// TwinCAT 3 PLC project Tc3_CRC
// Title: Tc3_CRC
// Company: RKe
// Author: Kim Robbens
// ProjectVersion: 0.0.0.2
// Description: CRC (Cyclic Redundancy Check) calculation with support for numerous standard CRC algorithms
// ProgramVersion: 3.1.4026.17
// libraries:
//   Tc2_Utilities, * (Beckhoff Automation GmbH)
//   Tc3_AlgoInterfaces, * (RKe)
// project tree:
//   DUTs/ E_CRC_Mode.TcDUT, E_CRC_Type.TcDUT, ST_CRC_Params.TcDUT, U_8BYTEARRAY.TcDUT
//   GVCs/ GVC_CRC.TcGVL
//   POUs/ CRC.TcPOU
//   Project Information/ F_GetCompany.TcPOU, F_GetTitle.TcPOU, F_GetVersion.TcPOU
//   Version/ Global_Version.TcGVL

// ---- DUTs/E_CRC_Mode.TcDUT
{attribute 'qualified_only'}
{attribute 'strict'}
{attribute 'to_string'}
TYPE E_CRC_Mode :
(
	CRC8	:= 0,
	CRC16 	:= 1,
	CRC24 	:= 2,
	CRC32 	:= 3,
	CRC40 	:= 4,
	CRC64 	:= 7
) BYTE;
END_TYPE

// ---- DUTs/E_CRC_Type.TcDUT
{attribute 'qualified_only'}
{attribute 'to_string'}
TYPE E_CRC_Type : (
    CRC_8_AUTOSAR,
    CRC_8_BLUETOOTH,
    CRC_8_CDMA2000,
    CRC_8_DARC,
    CRC_8_DVB_S2,
    CRC_8_GSM_A,
    CRC_8_GSM_B,
    CRC_8_HITAG,
    CRC_8_I_432_1,
    CRC_8_I_CODE,
    CRC_8_LTE,
    CRC_8_MAXIM_DOW,
    CRC_8_MIFARE_MAD,
    CRC_8_NRSC_5,
    CRC_8_OPENSAFETY,
    CRC_8_ROHC,
    CRC_8_SAE_J1850,
    CRC_8_SMBUS,
    CRC_8_TECH_3250,
    CRC_8_WCDMA,
    CRC_16_ARC,
    CRC_16_CDMA2000,
    CRC_16_CMS,
    CRC_16_DDS_110,
    CRC_16_DECT_R,
    CRC_16_DECT_X,
    CRC_16_DNP,
    CRC_16_EN_13757,
    CRC_16_GENIBUS,
    CRC_16_GSM,
    CRC_16_IBM_3740,
    CRC_16_IBM_SDLC,
    CRC_16_ISO_IEC_14443_3_A,
    CRC_16_KERMIT,
    CRC_16_LJ1200,
    CRC_16_MAXIM_DOW,
    CRC_16_MCRF4XX,
    CRC_16_MODBUS,
    CRC_16_NRSC_5,
    CRC_16_OPENSAFETY_A,
    CRC_16_OPENSAFETY_B,
    CRC_16_PROFIBUS,
    CRC_16_RIELLO,
    CRC_16_SPI_FUJITSU,
    CRC_16_T10_DIF,
    CRC_16_TELEDISK,
    CRC_16_TMS37157,
    CRC_16_UMTS,
    CRC_16_USB,
    CRC_16_XMODEM,
    CRC_24_BLE,
    CRC_24_FLEXRAY_A,
    CRC_24_FLEXRAY_B,
    CRC_24_INTERLAKEN,
    CRC_24_LTE_A,
    CRC_24_LTE_B,
    CRC_24_OPENPGP,
    CRC_24_OS_9,
    CRC_32_AIXM,
    CRC_32_AUTOSAR,
    CRC_32_BASE91_D,
    CRC_32_BZIP2,
    CRC_32_CD_ROM_EDC,
    CRC_32_CKSUM,
    CRC_32_ISCSI,
    CRC_32_ISO_HDLC,
    CRC_32_JAMCRC,
    CRC_32_MEF,
    CRC_32_MPEG_2,
    CRC_32_XFER,
    CRC_40_GSM,
    CRC_64_ECMA_182,
    CRC_64_GO_ISO,
    CRC_64_MS,
    CRC_64_WE,
    CRC_64_XZ,
	CRC_NO_OF_TYPES  		// end of enum list placeholder
)BYTE;
END_TYPE

// ---- DUTs/ST_CRC_Params.TcDUT
TYPE ST_CRC_Params :
STRUCT
    bitWidth      		: BYTE;
    polynomial       	: XWORD;
    initCRC       		: XWORD;
    reflectInitial      : BOOL;
    reflected     		: BOOL;
    xorOut     			: XWORD;
    check      			: XWORD;
    residue    			: XWORD;
END_STRUCT
END_TYPE

// ---- DUTs/U_8BYTEARRAY.TcDUT
TYPE U_8BYTEARRAY :
UNION
	byteArray					: ARRAY[0..7] OF BYTE;
	xword_						: XWORD;
	dword_						: ARRAY[0..1] OF DWORD;					
	word_						: ARRAY[0..3] OF WORD;					
END_UNION
END_TYPE

// ---- GVCs/GVC_CRC.TcGVL
{attribute 'qualified_only'}
VAR_GLOBAL CONSTANT
	CRCMasks 		: ARRAY[0..E_CRC_Mode.CRC64] OF XWORD 	:= [16#FF, 16#FFFF, 16#FFFFFF, 16#FFFFFFFF, 16#FFFFFFFFFF, 16#0, 16#0, 16#FFFFFFFFFFFFFFFF];
	CRCMsb			: ARRAY[0..E_CRC_Mode.CRC64] OF XWORD 	:= [16#80, 16#8000, 16#800000, 16#80000000, 16#8000000000, 16#0, 16#0, 16#8000000000000000]; 
	CRCShift		: ARRAY[0..E_CRC_Mode.CRC64] OF BYTE 	:= [0, 8, 16, 24, 32, 0, 0, 56];	
	referenceCheck	: ARRAY[1..9] OF BYTE := [16#31, 16#32, 16#33, 16#34, 16#35, 16#36, 16#37, 16#38, 16#39]; // Number 123456789  

	// CRC Type definition
	// source: https://reveng.sourceforge.io/crc-catalogue/all.htm
	CRC_Parameters : ARRAY[0..E_CRC_Type.CRC_NO_OF_TYPES] OF ST_CRC_Params := [
(* CRC_8_AUTOSAR *)      		(bitWidth := 8, polynomial := 16#2F, initCRC := 16#FF, reflectInitial := FALSE, reflected := FALSE, XorOut := 16#FF, Check := 16#DF, Residue := 16#42),
(* CRC_8_BLUETOOTH *)    		(bitWidth := 8, polynomial := 16#A7, initCRC := 16#00, reflectInitial := FALSE, reflected := TRUE,  XorOut := 16#00, Check := 16#26, Residue := 16#00),
(* CRC_8_CDMA2000 *)     		(bitWidth := 8, polynomial := 16#9B, initCRC := 16#FF, reflectInitial := FALSE, reflected := FALSE, XorOut := 16#00, Check := 16#DA, Residue := 16#00),
(* CRC_8_DARC *)         		(bitWidth := 8, polynomial := 16#39, initCRC := 16#00, reflectInitial := FALSE, reflected := TRUE,  XorOut := 16#00, Check := 16#15, Residue := 16#00),
(* CRC_8_DVB_S2 *)       		(bitWidth := 8, polynomial := 16#D5, initCRC := 16#00, reflectInitial := FALSE, reflected := FALSE, XorOut := 16#00, Check := 16#BC, Residue := 16#00),
(* CRC_8_GSM_A *)        		(bitWidth := 8, polynomial := 16#1D, initCRC := 16#00, reflectInitial := FALSE, reflected := FALSE, XorOut := 16#00, Check := 16#37, Residue := 16#00),
(* CRC_8_GSM_B *)        		(bitWidth := 8, polynomial := 16#49, initCRC := 16#00, reflectInitial := FALSE, reflected := FALSE, XorOut := 16#FF, Check := 16#94, Residue := 16#53),
(* CRC_8_HITAG *)        		(bitWidth := 8, polynomial := 16#1D, initCRC := 16#FF, reflectInitial := FALSE, reflected := FALSE, XorOut := 16#00, Check := 16#B4, Residue := 16#00),
(* CRC_8_I_432_1 *)      		(bitWidth := 8, polynomial := 16#07, initCRC := 16#00, reflectInitial := FALSE, reflected := FALSE, XorOut := 16#55, Check := 16#A1, Residue := 16#AC),
(* CRC_8_I_CODE *)       		(bitWidth := 8, polynomial := 16#1D, initCRC := 16#FD, reflectInitial := FALSE, reflected := FALSE, XorOut := 16#00, Check := 16#7E, Residue := 16#00),
(* CRC_8_LTE *)          		(bitWidth := 8, polynomial := 16#9B, initCRC := 16#00, reflectInitial := FALSE, reflected := FALSE, XorOut := 16#00, Check := 16#EA, Residue := 16#00),
(* CRC_8_MAXIM_DOW *)    		(bitWidth := 8, polynomial := 16#31, initCRC := 16#00, reflectInitial := FALSE, reflected := TRUE,  XorOut := 16#00, Check := 16#A1, Residue := 16#00),
(* CRC_8_MIFARE_MAD *)   		(bitWidth := 8, polynomial := 16#1D, initCRC := 16#C7, reflectInitial := FALSE, reflected := FALSE, XorOut := 16#00, Check := 16#99, Residue := 16#00),
(* CRC_8_NRSC_5 *)       		(bitWidth := 8, polynomial := 16#31, initCRC := 16#FF, reflectInitial := FALSE, reflected := FALSE, XorOut := 16#00, Check := 16#F7, Residue := 16#00),
(* CRC_8_OPENSAFETY *)   		(bitWidth := 8, polynomial := 16#2F, initCRC := 16#00, reflectInitial := FALSE, reflected := FALSE, XorOut := 16#00, Check := 16#3E, Residue := 16#00),
(* CRC_8_ROHC *)         		(bitWidth := 8, polynomial := 16#07, initCRC := 16#FF, reflectInitial := FALSE, reflected := TRUE,  XorOut := 16#00, Check := 16#D0, Residue := 16#00),
(* CRC_8_SAE_J1850 *)    		(bitWidth := 8, polynomial := 16#1D, initCRC := 16#FF, reflectInitial := FALSE, reflected := FALSE, XorOut := 16#FF, Check := 16#4B, Residue := 16#C4),
(* CRC_8_SMBUS *)        		(bitWidth := 8, polynomial := 16#07, initCRC := 16#00, reflectInitial := FALSE, reflected := FALSE, XorOut := 16#00, Check := 16#F4, Residue := 16#00),
(* CRC_8_TECH_3250 *)    		(bitWidth := 8, polynomial := 16#1D, initCRC := 16#FF, reflectInitial := FALSE, reflected := TRUE,  XorOut := 16#00, Check := 16#97, Residue := 16#00),
(* CRC_8_WCDMA *)        		(bitWidth := 8, polynomial := 16#9B, initCRC := 16#00, reflectInitial := FALSE, reflected := TRUE,  XorOut := 16#00, Check := 16#25, Residue := 16#00),
(* CRC_16_ARC *)                (bitWidth := 16, polynomial := 16#8005, initCRC := 16#0000, reflectInitial := FALSE, reflected := TRUE,  XorOut := 16#0000, Check := 16#BB3D, Residue := 16#0000),
(* CRC_16_CDMA2000 *)           (bitWidth := 16, polynomial := 16#C867, initCRC := 16#FFFF, reflectInitial := FALSE, reflected := FALSE, XorOut := 16#0000, Check := 16#4C06, Residue := 16#0000),
(* CRC_16_CMS *)                (bitWidth := 16, polynomial := 16#8005, initCRC := 16#FFFF, reflectInitial := FALSE, reflected := FALSE, XorOut := 16#0000, Check := 16#AEE7, Residue := 16#0000),
(* CRC_16_DDS_110 *)            (bitWidth := 16, polynomial := 16#8005, initCRC := 16#800D, reflectInitial := FALSE, reflected := FALSE, XorOut := 16#0000, Check := 16#9ECF, Residue := 16#0000),
(* CRC_16_DECT_R *)             (bitWidth := 16, polynomial := 16#0589, initCRC := 16#0000, reflectInitial := FALSE, reflected := FALSE, XorOut := 16#0001, Check := 16#007E, Residue := 16#0589),
(* CRC_16_DECT_X *)             (bitWidth := 16, polynomial := 16#0589, initCRC := 16#0000, reflectInitial := FALSE, reflected := FALSE, XorOut := 16#0000, Check := 16#007F, Residue := 16#0000),
(* CRC_16_DNP *)                (bitWidth := 16, polynomial := 16#3D65, initCRC := 16#0000, reflectInitial := FALSE, reflected := TRUE,  XorOut := 16#FFFF, Check := 16#EA82, Residue := 16#66C5),
(* CRC_16_EN_13757 *)           (bitWidth := 16, polynomial := 16#3D65, initCRC := 16#0000, reflectInitial := FALSE, reflected := FALSE, XorOut := 16#FFFF, Check := 16#C2B7, Residue := 16#A366),
(* CRC_16_GENIBUS *)            (bitWidth := 16, polynomial := 16#1021, initCRC := 16#FFFF, reflectInitial := FALSE, reflected := FALSE, XorOut := 16#FFFF, Check := 16#D64E, Residue := 16#1D0F),
(* CRC_16_GSM *)                (bitWidth := 16, polynomial := 16#1021, initCRC := 16#0000, reflectInitial := FALSE, reflected := FALSE, XorOut := 16#FFFF, Check := 16#CE3C, Residue := 16#1D0F),
(* CRC_16_IBM_3740 *)           (bitWidth := 16, polynomial := 16#1021, initCRC := 16#FFFF, reflectInitial := FALSE, reflected := FALSE, XorOut := 16#0000, Check := 16#29B1, Residue := 16#0000),
(* CRC_16_IBM_SDLC *)           (bitWidth := 16, polynomial := 16#1021, initCRC := 16#FFFF, reflectInitial := FALSE, reflected := TRUE,  XorOut := 16#FFFF, Check := 16#906E, Residue := 16#F0B8),
(* CRC_16_ISO_IEC_14443_3_A *)  (bitWidth := 16, polynomial := 16#1021, initCRC := 16#C6C6, reflectInitial := TRUE,  reflected := TRUE,  XorOut := 16#0000, Check := 16#BF05, Residue := 16#0000),
(* CRC_16_KERMIT *)             (bitWidth := 16, polynomial := 16#1021, initCRC := 16#0000, reflectInitial := FALSE, reflected := TRUE,  XorOut := 16#0000, Check := 16#2189, Residue := 16#0000),
(* CRC_16_LJ1200 *)             (bitWidth := 16, polynomial := 16#6F63, initCRC := 16#0000, reflectInitial := FALSE, reflected := FALSE, XorOut := 16#0000, Check := 16#BDF4, Residue := 16#0000),
(* CRC_16_MAXIM_DOW *)          (bitWidth := 16, polynomial := 16#8005, initCRC := 16#0000, reflectInitial := FALSE, reflected := TRUE,  XorOut := 16#FFFF, Check := 16#44C2, Residue := 16#B001),
(* CRC_16_MCRF4XX *)            (bitWidth := 16, polynomial := 16#1021, initCRC := 16#FFFF, reflectInitial := FALSE, reflected := TRUE,  XorOut := 16#0000, Check := 16#6F91, Residue := 16#0000),
(* CRC_16_MODBUS *)             (bitWidth := 16, polynomial := 16#8005, initCRC := 16#FFFF, reflectInitial := FALSE, reflected := TRUE,  XorOut := 16#0000, Check := 16#4B37, Residue := 16#0000),
(* CRC_16_NRSC_5 *)             (bitWidth := 16, polynomial := 16#080B, initCRC := 16#FFFF, reflectInitial := FALSE, reflected := TRUE,  XorOut := 16#0000, Check := 16#A066, Residue := 16#0000),
(* CRC_16_OPENSAFETY_A *)       (bitWidth := 16, polynomial := 16#5935, initCRC := 16#0000, reflectInitial := FALSE, reflected := FALSE, XorOut := 16#0000, Check := 16#5D38, Residue := 16#0000),
(* CRC_16_OPENSAFETY_B *)       (bitWidth := 16, polynomial := 16#755B, initCRC := 16#0000, reflectInitial := FALSE, reflected := FALSE, XorOut := 16#0000, Check := 16#20FE, Residue := 16#0000),
(* CRC_16_PROFIBUS *)           (bitWidth := 16, polynomial := 16#1DCF, initCRC := 16#FFFF, reflectInitial := FALSE, reflected := FALSE, XorOut := 16#FFFF, Check := 16#A819, Residue := 16#E394),
(* CRC_16_RIELLO *)             (bitWidth := 16, polynomial := 16#1021, initCRC := 16#B2AA, reflectInitial := TRUE,  reflected := TRUE,  XorOut := 16#0000, Check := 16#63D0, Residue := 16#0000),
(* CRC_16_SPI_FUJITSU *)        (bitWidth := 16, polynomial := 16#1021, initCRC := 16#1D0F, reflectInitial := FALSE, reflected := FALSE, XorOut := 16#0000, Check := 16#E5CC, Residue := 16#0000),
(* CRC_16_T10_DIF *)            (bitWidth := 16, polynomial := 16#8BB7, initCRC := 16#0000, reflectInitial := FALSE, reflected := FALSE, XorOut := 16#0000, Check := 16#D0DB, Residue := 16#0000),
(* CRC_16_TELEDISK *)           (bitWidth := 16, polynomial := 16#A097, initCRC := 16#0000, reflectInitial := FALSE, reflected := FALSE, XorOut := 16#0000, Check := 16#0FB3, Residue := 16#0000),
(* CRC_16_TMS37157 *)           (bitWidth := 16, polynomial := 16#1021, initCRC := 16#89EC, reflectInitial := TRUE,  reflected := TRUE,  XorOut := 16#0000, Check := 16#26B1, Residue := 16#0000),
(* CRC_16_UMTS *)               (bitWidth := 16, polynomial := 16#8005, initCRC := 16#0000, reflectInitial := FALSE, reflected := FALSE, XorOut := 16#0000, Check := 16#FEE8, Residue := 16#0000),
(* CRC_16_USB *)                (bitWidth := 16, polynomial := 16#8005, initCRC := 16#FFFF, reflectInitial := FALSE, reflected := TRUE,  XorOut := 16#FFFF, Check := 16#B4C8, Residue := 16#B001),
(* CRC_16_XMODEM *)             (bitWidth := 16, polynomial := 16#1021, initCRC := 16#0000, reflectInitial := FALSE, reflected := FALSE, XorOut := 16#0000, Check := 16#31C3, Residue := 16#0000),
(* CRC_24_BLE *)          		(bitWidth := 24, polynomial := 16#00065B,   initCRC := 16#555555,   reflectInitial := TRUE,  reflected := TRUE,  XorOut := 16#000000,   Check := 16#C25A56,   Residue := 16#000000),
(* CRC_24_FLEXRAY_A *)    		(bitWidth := 24, polynomial := 16#5D6DCB,   initCRC := 16#FEDCBA,   reflectInitial := FALSE, reflected := FALSE, XorOut := 16#000000,   Check := 16#7979BD,   Residue := 16#000000),
(* CRC_24_FLEXRAY_B *)    		(bitWidth := 24, polynomial := 16#5D6DCB,   initCRC := 16#ABCDEF,   reflectInitial := FALSE, reflected := FALSE, XorOut := 16#000000,   Check := 16#1F23B8,   Residue := 16#000000),
(* CRC_24_INTERLAKEN *)   		(bitWidth := 24, polynomial := 16#328B63,   initCRC := 16#FFFFFF,   reflectInitial := FALSE, reflected := FALSE, XorOut := 16#FFFFFF,   Check := 16#B4F3E6,   Residue := 16#144E63),
(* CRC_24_LTE_A *)        		(bitWidth := 24, polynomial := 16#864CFB,   initCRC := 16#000000,   reflectInitial := FALSE, reflected := FALSE, XorOut := 16#000000,   Check := 16#CDE703,   Residue := 16#000000),
(* CRC_24_LTE_B *)        		(bitWidth := 24, polynomial := 16#800063,   initCRC := 16#000000,   reflectInitial := FALSE, reflected := FALSE, XorOut := 16#000000,   Check := 16#23EF52,   Residue := 16#000000),
(* CRC_24_OPENPGP *)      		(bitWidth := 24, polynomial := 16#864CFB,   initCRC := 16#B704CE,   reflectInitial := FALSE, reflected := FALSE, XorOut := 16#000000,   Check := 16#21CF02,   Residue := 16#000000),
(* CRC_24_OS_9 *)         		(bitWidth := 24, polynomial := 16#800063,   initCRC := 16#FFFFFF,   reflectInitial := FALSE, reflected := FALSE, XorOut := 16#FFFFFF,   Check := 16#200FA5,   Residue := 16#800FE3),
(* CRC_32_AIXM *)         		(bitWidth := 32, polynomial := 16#814141AB, initCRC := 16#00000000, reflectInitial := FALSE, reflected := FALSE, XorOut := 16#00000000, Check := 16#3010BF7F, Residue := 16#00000000),
(* CRC_32_AUTOSAR *)      		(bitWidth := 32, polynomial := 16#F4ACFB13, initCRC := 16#FFFFFFFF, reflectInitial := FALSE, reflected := TRUE,  XorOut := 16#FFFFFFFF, Check := 16#1697D06A, Residue := 16#904CDDBF),
(* CRC_32_BASE91_D *)     		(bitWidth := 32, polynomial := 16#A833982B, initCRC := 16#FFFFFFFF, reflectInitial := FALSE, reflected := TRUE,  XorOut := 16#FFFFFFFF, Check := 16#87315576, Residue := 16#45270551),
(* CRC_32_BZIP2 *)        		(bitWidth := 32, polynomial := 16#04C11DB7, initCRC := 16#FFFFFFFF, reflectInitial := FALSE, reflected := FALSE, XorOut := 16#FFFFFFFF, Check := 16#FC891918, Residue := 16#C704DD7B),
(* CRC_32_CD_ROM_EDC *)   		(bitWidth := 32, polynomial := 16#8001801B, initCRC := 16#00000000, reflectInitial := FALSE, reflected := TRUE,  XorOut := 16#00000000, Check := 16#6EC2EDC4, Residue := 16#00000000),
(* CRC_32_CKSUM *)        		(bitWidth := 32, polynomial := 16#04C11DB7, initCRC := 16#00000000, reflectInitial := FALSE, reflected := FALSE, XorOut := 16#FFFFFFFF, Check := 16#765E7680, Residue := 16#C704DD7B),
(* CRC_32_ISCSI *)        		(bitWidth := 32, polynomial := 16#1EDC6F41, initCRC := 16#FFFFFFFF, reflectInitial := FALSE, reflected := TRUE,  XorOut := 16#FFFFFFFF, Check := 16#E3069283, Residue := 16#B798B438),
(* CRC_32_ISO_HDLC *)     		(bitWidth := 32, polynomial := 16#04C11DB7, initCRC := 16#FFFFFFFF, reflectInitial := FALSE, reflected := TRUE,  XorOut := 16#FFFFFFFF, Check := 16#CBF43926, Residue := 16#DEBB20E3),
(* CRC_32_JAMCRC *)       		(bitWidth := 32, polynomial := 16#04C11DB7, initCRC := 16#FFFFFFFF, reflectInitial := FALSE, reflected := TRUE,  XorOut := 16#00000000, Check := 16#340BC6D9, Residue := 16#00000000),
(* CRC_32_MEF *)          		(bitWidth := 32, polynomial := 16#741B8CD7, initCRC := 16#FFFFFFFF, reflectInitial := FALSE, reflected := TRUE,  XorOut := 16#00000000, Check := 16#D2C22F51, Residue := 16#00000000),
(* CRC_32_MPEG_2 *)       		(bitWidth := 32, polynomial := 16#04C11DB7, initCRC := 16#FFFFFFFF, reflectInitial := FALSE, reflected := FALSE, XorOut := 16#00000000, Check := 16#0376E6E7, Residue := 16#00000000),
(* CRC_32_XFER *)         		(bitWidth := 32, polynomial := 16#000000AF, initCRC := 16#00000000, reflectInitial := FALSE, reflected := FALSE, XorOut := 16#00000000, Check := 16#BD0BE338, Residue := 16#00000000),
(* CRC_40_GSM *)        	    (bitWidth := 40, polynomial := 16#0004820009, initCRC := 16#0000000000, reflectInitial := FALSE, reflected := FALSE, XorOut := 16#FFFFFFFFFF, Check := 16#D4164FC646, Residue := 16#C4FF8071FF),
(* CRC_64_ECMA_182 *)   		(bitWidth := 64, polynomial := 16#42F0E1EBA9EA3693, initCRC := 16#0000000000000000, reflectInitial := FALSE, reflected := FALSE, XorOut := 16#0000000000000000, Check := 16#6C40DF5F0B497347, Residue := 16#0000000000000000),
(* CRC_64_GO_ISO *)     		(bitWidth := 64, polynomial := 16#000000000000001B, initCRC := 16#FFFFFFFFFFFFFFFF, reflectInitial := FALSE, reflected := TRUE,  XorOut := 16#FFFFFFFFFFFFFFFF, Check := 16#B90956C775A41001, Residue := 16#5300000000000000),
(* CRC_64_MS *)         		(bitWidth := 64, polynomial := 16#259C84CBA6426349, initCRC := 16#FFFFFFFFFFFFFFFF, reflectInitial := FALSE, reflected := TRUE,  XorOut := 16#0000000000000000, Check := 16#75D4B74F024ECEEA, Residue := 16#0000000000000000),
(* CRC_64_WE *)         		(bitWidth := 64, polynomial := 16#42F0E1EBA9EA3693, initCRC := 16#FFFFFFFFFFFFFFFF, reflectInitial := FALSE, reflected := FALSE, XorOut := 16#FFFFFFFFFFFFFFFF, Check := 16#62EC59E3F1A4F00A, Residue := 16#FCACBEBD5931A992),
(* CRC_64_XZ *)         		(bitWidth := 64, polynomial := 16#42F0E1EBA9EA3693, initCRC := 16#FFFFFFFFFFFFFFFF, reflectInitial := FALSE, reflected := TRUE,  XorOut := 16#FFFFFFFFFFFFFFFF, Check := 16#995DC9BBDF1939FA, Residue := 16#49958C9ABD7D353F)
    ];
END_VAR

// ---- Version/Global_Version.TcGVL
{attribute 'TcGenerated'}
{attribute 'no-analysis'}
{attribute 'linkalways'}
// This function has been automatically generated from the project information.
VAR_GLOBAL CONSTANT
	{attribute 'const_non_replaced'}
	stLibVersion_Tc3_CRC : ST_LibVersion := (iMajor := 0, iMinor := 0, iBuild := 0, iRevision := 2, nFlags := 0, sVersion := '0.0.0.2');
END_VAR

// ---- POUs/CRC.TcPOU
{attribute 'no_explicit_call' := 'do not call this POU directly'} 
FUNCTION_BLOCK CRC IMPLEMENTS Tc3_AlgoInterfaces.IDigest
VAR
	// values are precalulated in FB_Init 
	CRCTableInitialized				: BOOL;
	// Precalcated lookup table
	CRC_Table 						: ARRAY[0..TABLESIZE-1] OF XWORD;
	// Current crc
	currentCrc						: XWORD;					
	// CRC parameters
	_crcType						: E_CRC_TYPE;
	_polynomial						: XWORD;		// polynomial 
	_polynomial_					: XWORD;		// reflected polynomial 
	_bitWidth						: BYTE;
	_initCrc						: XWORD;
	_reflectInitial					: BOOL;
	_reflected						: BOOL;
	_xorOut							: XWORD;
	_check							: XWORD;
	_residue						: XWORD;
	// internal 
	isInitialReflected				: BOOL;
END_VAR
VAR CONSTANT
	// Maximum size of the lookup table (no of byte values)
	TABLESIZE						: UINT := 256;
END_VAR

// use compute method

PROPERTY algorithm : STRING
GET
algorithm := TO_STRING(_crcType);
END_GET
END_PROPERTY

// Computes CRC using a standard (non-reflected) lookup table
METHOD PRIVATE computeNormal : XWORD
VAR_INPUT
    pData 						: POINTER TO BYTE;
	dataSize					: DWORD;
END_VAR
VAR
	pByte 						: POINTER TO BYTE;
	bByte						: BYTE;
	mode 						: BYTE;
	i 							: DWORD;
	lookupIndex					: BYTE;
END_VAR
mode					:= TO_BYTE(_bitWidth / 8) - 1;
computeNormal 			:= currentCrc;

pByte					:= pData;
FOR i := 0 TO dataSize - 1 DO
	bByte				:= pByte^;
	pByte				:= pByte + 1;
	lookupIndex			:= TO_BYTE(SHR(computeNormal, GVC_CRC.crcShift[mode]) XOR bByte);	
	IF (mode = E_CRC_Mode.CRC8)	THEN
		computeNormal	:= CRC_Table[lookupIndex];
	ELSE
		computeNormal	:= SHL(computeNormal, 8) XOR CRC_Table[lookupIndex];
	END_IF
	computeNormal		:= computeNormal AND GVC_CRC.crcMasks[mode]; 
END_FOR
END_METHOD

// Computes CRC using a reflected lookup table
METHOD PRIVATE computeReflected : XWORD
VAR_INPUT
    pData 						: POINTER TO BYTE;
	dataSize					: DWORD;
END_VAR
VAR
	pByte 						: POINTER TO BYTE;
	bByte						: BYTE;
	i 							: DWORD;
	lookupIndex					: BYTE;
END_VAR
computeReflected 		:= currentCrc;

pByte					:= pData;
FOR i := 0 TO dataSize - 1 DO
	bByte				:= pByte^;
	pByte				:= pByte + 1;
	lookupIndex			:= TO_BYTE((computeReflected XOR bByte) AND GVC_CRC.crcMasks[0]);
	computeReflected	:= SHR(computeReflected, 8) XOR CRC_Table[lookupIndex];
END_FOR
END_METHOD

METHOD FB_Init: BOOL
VAR_INPUT
    bInitRetains				: BOOL; // TRUE: the retain variables are initialized (reset warm / reset cold)
    bInCopyCode					: BOOL; // TRUE: the instance will be copied to the copy code afterward (online change)   
	crcType						: E_CRC_TYPE;
END_VAR
// Pass to the local init
reconfigure(crcType);
END_METHOD

(* Finalize the input and return any number of output bytes.*)
METHOD finalize
VAR_IN_OUT
	out					: ARRAY [*] OF BYTE;
END_VAR
VAR
	byteVal, mode		: BYTE;
	i, j, ub			: DINT;
END_VAR
// Final xor and mask
mode					:= TO_BYTE(_bitWidth / 8) - 1;
currentCrc				:= (currentCrc XOR _xorOut) AND GVC_CRC.crcMasks[mode];

j 	:= LOWER_BOUND(out, 1);
ub 	:= UPPER_BOUND(out, 1);
FOR i := 0 TO GVC_CRC.CRC_Parameters[_crcType].bitWidth / 8 - 1 DO
	IF i > ub THEN // in case the wrong crc result container was passed
		EXIT;
	ELSE
		byteVal	:= TO_BYTE(SHR(currentCrc, i * 8));
		//byteVal := TO_BYTE(SHR(byteVal, 56)
		out[i]  := byteVal; // TO_BYTE(SHR(SHL(currentCrc, i * 8), 56));
	END_IF
END_FOR
END_METHOD

// Generates a standard CRC lookup table
METHOD PRIVATE generateNormalCRCTable : BOOL
VAR
	mode					: BYTE;
	crc						: XWORD;
	i, j					: UINT; 
END_VAR
generateNormalCRCTable := FALSE;
mode := (_bitWidth / 8) - 1;

FOR i := 0 TO TABLESIZE - 1 DO
	crc			:= (SHL(TO___XWORD(i), GVC_CRC.CRCShift[mode])) AND GVC_CRC.CRCMasks[mode];
	FOR j := 0 TO 7 DO
		IF (crc AND GVC_CRC.CRCMsb[Mode]) = 0 THEN
			crc :=  SHL(crc, 1); 
		ELSE
			crc := SHL(crc, 1) XOR _polynomial;
		END_IF
		crc		:= crc AND GVC_CRC.CRCMasks[mode];
  	END_FOR
	CRC_Table[i]:= crc;
END_FOR
generateNormalCRCTable := TRUE;
END_METHOD

// Generates a reflected CRC lookup table
METHOD PRIVATE generateReflectedCRCTable : BOOL
VAR
	mode					: BYTE;
	crc						: XWORD;
	i, j					: UINT; 
END_VAR
generateReflectedCRCTable := FALSE;	 
mode := (_bitWidth / 8) - 1;

FOR i := 0 TO TABLESIZE - 1 DO
	crc			:= i;
	FOR j := 0 TO 7 DO
		IF (crc AND 16#1) = 0 THEN
			crc :=  SHR(crc, 1); 
		ELSE
			crc := SHR(crc, 1) XOR _polynomial_;
		END_IF
		crc		:= crc AND GVC_CRC.CRCMasks[mode];
  	END_FOR
	CRC_Table[i]:= crc;
END_FOR
generateReflectedCRCTable := TRUE;
END_METHOD

METHOD init
// Reset the crc to the configured initial value 
currentCrc 			:= _initCrc;
isInitialReflected		:= FALSE;
END_METHOD

// Reconfigures and initializes the CRC table in function of chosen CRC Type
METHOD reconfigure : bool
VAR_INPUT
	crcType						: E_CRC_TYPE;
END_VAR
// CRC parameters
_crcType				:= crcType;
_bitWidth				:= GVC_CRC.CRC_Parameters[_crcType].bitWidth;
_polynomial				:= GVC_CRC.CRC_Parameters[_crcType].polynomial; 
_polynomial_			:= reflectBits(_polynomial, _bitWidth);
_initCrc				:= GVC_CRC.CRC_Parameters[_crcType].initCRC;
_reflectInitial			:= GVC_CRC.CRC_Parameters[_crcType].reflectInitial;
_reflected				:= GVC_CRC.CRC_Parameters[_crcType].reflected;
_xorOut					:= GVC_CRC.CRC_Parameters[_crcType].xorOut;
_check					:= GVC_CRC.CRC_Parameters[_crcType].check;
_residue				:= GVC_CRC.CRC_Parameters[_crcType].residue;

// Build CRC table
CRCTableInitialized := FALSE;
IF GVC_CRC.CRC_Parameters[_crcType].polynomial > 0 THEN		// Valid polynomial
	IF _reflected			THEN
		CRCTableInitialized	:= generateReflectedCRCTable();
	ELSE
		CRCTableInitialized	:= generateNormalCRCTable();
	END_IF
END_IF

// initialize 
init();
END_METHOD

// Reflects the bit order of a value
METHOD PRIVATE reflectBits		: XWORD
VAR_INPUT
	value 						: XWORD;
	bitWidth					: BYTE;
END_VAR
VAR
	i							: BYTE;
	shrValue					: XWORD;
	andBit						: XWORD;
END_VAR
reflectBits 		:= 16#0;
shrValue 		:= value;
andBit 			:= shrValue AND 16#1;
reflectBits 		:= reflectBits + andBit;
FOR i := 1 TO bitWidth - 1 DO
	reflectBits 	:= SHL(reflectBits,1);
	shrValue 	:= SHR(shrValue,1);
	andBit 		:= shrValue AND 16#1;
	reflectBits 	:= reflectBits + andBit;
END_FOR
END_METHOD

(* Add input, depending on the algorithm this could be called any number of times.*)
METHOD update
VAR_INPUT
	input						: POINTER TO BYTE;
	input_len					: DWORD;
END_VAR
IF _reflectInitial		AND NOT 
	isInitialReflected		THEN
	currentCrc			:= reflectBits(currentCrc, _bitWidth);
	isInitialReflected		:= TRUE;
END_IF

IF _reflected			THEN
	currentCrc := computeReflected(input, input_len);
ELSE
	currentCrc := computeNormal(input, input_len);
END_IF
END_METHOD

END_FUNCTION_BLOCK

// ---- Project Information/F_GetCompany.TcPOU
// This function has been automatically generated from the project information.
{attribute 'signature_flag' := '1073741824'}
{attribute 'TcGenerated'}
{attribute 'no-analysis'}
FUNCTION F_GetCompany : WSTRING
VAR_INPUT
	
END_VAR

F_GetCompany := "Kim Robbens";

END_FUNCTION

// ---- Project Information/F_GetTitle.TcPOU
// This function has been automatically generated from the project information.
{attribute 'signature_flag' := '1073741824'}
{attribute 'TcGenerated'}
{attribute 'no-analysis'}
FUNCTION F_GetTitle : WSTRING
VAR_INPUT
	
END_VAR

F_GetTitle := "Tc3_CRC";

END_FUNCTION

// ---- Project Information/F_GetVersion.TcPOU
// This function has been automatically generated from the project information.
{attribute 'signature_flag' := '1073741824'}
{attribute 'TcGenerated'}
{attribute 'no-analysis'}
FUNCTION F_GetVersion : ST_LibVersion
VAR_INPUT
	
END_VAR

F_GetVersion.iMajor := 0;
F_GetVersion.iMinor := 0;
F_GetVersion.iBuild := 0;
F_GetVersion.iRevision := 1;
F_GetVersion.sVersion := '0.0.0.1';
F_GetVersion.nFlags := 0;

END_FUNCTION
